TYPE T_CodeRSKU : STRING[9];
END_TYPE

(* stored: Version 1.1.0.1
   DUT T_CodeRSKU: Id {91780bfa-c3d8-4563-ad05-a5565361cf58} *)
